(* IEC 61131-3 sources: dynamics/test, 21 files *)

(* ---- DeadbeatTest.st ---- *)
USING Simatic.Ax.Dynamics;
USING AxUnit;
USING System.Math;
NAMESPACE MyTest

    FUNCTION PT1 : LREAL
        VAR_INPUT
            t : LREAL;
            value : LREAL;
            output : LREAL;
            k : LREAL;
            t0 : LREAL;
        END_VAR
        PT1 := k * value + (output - k * value) * Exp(-1.0 * t / t0);
    END_FUNCTION

    {TestFixture}
    CLASS DeadbeatTest EXTENDS GlobalTest
        VAR
            controller : PT1_DeadbeatController;
        END_VAR

        {Test(k := 1, t0 := 1, output := 0, input := 0)}
        {Test(k := 1, t0 := 1, output := 0, input := 1)}
        {Test(k := 1, t0 := 1, output := 1, input := 0)}
        {Test(k := 1, t0 := 1, output := -78.5, input := 2.3)}
        {Test(k := 3.7, t0 := 5.8, output := -78.5, input := 2.3)}
        {Test(k := 107, t0 := 0.23, output := 10, input := 11)}
        METHOD PUBLIC Test
            VAR_INPUT
                k : LREAL;
                t0 : LREAL;
                output : LREAL;
                input : LREAL;
            END_VAR
            controller.SetK(k);
            controller.SetPeriods(oneSecondProvider.seconds, t0);
            Assert.Tolerated(input, PT1(oneSecondProvider.seconds, controller.Next(output, input), output, k, t0), TOLERANCE);
        END_METHOD
    END_CLASS
END_NAMESPACE

(* ---- Tolerated.st ---- *)
USING System.Math;
NAMESPACE AxUnit.Assert
    FUNCTION Tolerated
        VAR_INPUT
            expected : LREAL;
            actual : LREAL;
            tolerance : LREAL;
        END_VAR
        GreaterOrEqual(actual, expected - tolerance);
        LessOrEqual   (actual, expected + tolerance);
    END_FUNCTION
END_NAMESPACE

(* ---- AmplifierTest.st ---- *)
USING Simatic.Ax.Dynamics;

NAMESPACE MyTest
    {TestFixture}
    CLASS AmplifierTest EXTENDS GlobalTest

        VAR
            amplifier                   : Amplifier;
            value                       : ConstantSignal;
            expected                    : ConstantSignal;
        END_VAR

        // Amplifier
        {Test(k := 0, valueStepheight := 2.75)}
        {Test(k := 1, valueStepheight := 2.83)}
        {Test(k := 7.2, valueStepheight := 9.329)}
        {Test(k := 0.32, valueStepheight := 25.67)}
        METHOD PUBLIC Test
            VAR_INPUT
                k : LREAL;
                valueStepheight : LREAL;
            END_VAR
            amplifier.SetK(k);
            value.SetOutput(valueStepheight);
            expected.SetOutput(k * valueStepheight);
            THIS.AssertDynamic(expected, amplifier, value);
        END_METHOD

    END_CLASS
END_NAMESPACE

(* ---- BangBangTest.st ---- *)
USING Simatic.Ax.Dynamics;
USING AxUnit;

NAMESPACE MyTest
    {TestFixture}
    CLASS BangBangTest EXTENDS GlobalTest
        VAR
            controller : BangBangController;
        END_VAR

        // value0, value1, value2 and value3 are inside hysteresis
        {Test(input := 0, hysteresis := 1, output := FALSE, value0 := 0, value1 := 0, value2 := 0, value3 := 0)}
        {Test(input := 0, hysteresis := 1, output :=  TRUE, value0 := 0, value1 := 0, value2 := 0, value3 := 0)}
        {Test(input := 0, hysteresis := 1, output :=  TRUE, value0 := 0, value1 := -1, value2 := 1, value3 := 0.5)}
        {Test(input := 0, hysteresis := 10, output := FALSE, value0 := 2, value1 := -3, value2 := 5.7, value3 := -3.9)}
        {Test(input := 0, hysteresis := 83, output := TRUE, value0 := 20, value1 := -82.9, value2 := -83, value3 := 1.7)}
        METHOD PUBLIC TestWithinHysteresis
            VAR_INPUT
                input : LREAL;
                hysteresis: LREAL;
                output : BOOL;
                value0 : LREAL;
                value1 : LREAL;
                value2 : LREAL;
                value3 : LREAL;
            END_VAR
            controller.SetInput(input);
            controller.hysteresis := hysteresis;
            controller.SetOutput(output);
            Assert.Equal(controller.Next(value0), output);
            Assert.Equal(controller.Next(value1), output);
            Assert.Equal(controller.Next(value2), output);
            Assert.Equal(controller.Next(value3), output);
        END_METHOD

        // value is outside hysteresis
        {Test(input := 0,   hysteresis := 1,    heatingMode :=  TRUE, value := 2, expected := FALSE)}
        {Test(input := 0,   hysteresis := 1,    heatingMode := FALSE, value := 2, expected := TRUE)}
        {Test(input := 0,   hysteresis := 1,    heatingMode :=  TRUE, value := -2, expected := TRUE)}
        {Test(input := 0,   hysteresis := 1,    heatingMode := FALSE, value := -2, expected := FALSE)}
        {Test(input := 45,  hysteresis := 10,   heatingMode := FALSE, value := 34, expected := FALSE)}
        {Test(input := -3,  hysteresis := 0.1,  heatingMode := FALSE, value := -8, expected := FALSE)}
        {Test(input :=-107.59, hysteresis := 0, heatingMode := FALSE, value := -107.591, expected := FALSE)}
        {Test(input := 36.8, hysteresis := 2.5, heatingMode := FALSE, value := 31.8, expected := FALSE)}
        {Test(input := 45,  hysteresis := 10,   heatingMode :=  TRUE, value := 34, expected := TRUE)}
        {Test(input := -3,  hysteresis := 0.1,  heatingMode :=  TRUE, value := -8, expected := TRUE)}
        {Test(input :=-107.59, hysteresis := 0, heatingMode :=  TRUE, value := -107.591, expected := TRUE)}
        {Test(input := 36.8, hysteresis := 2.5, heatingMode :=  TRUE, value := 31.8, expected := TRUE)}
        {Test(input := 45,  hysteresis := 10,   heatingMode :=  TRUE, value := 56, expected := FALSE)}
        {Test(input := -3,  hysteresis := 0.1,  heatingMode :=  TRUE, value := -2, expected := FALSE)}
        {Test(input :=-107.59, hysteresis := 0, heatingMode :=  TRUE, value := -107.58, expected := FALSE)}
        {Test(input := 36.8, hysteresis := 2.5, heatingMode :=  TRUE, value := 41.8, expected := FALSE)}
        {Test(input := 45,  hysteresis := 10,   heatingMode := FALSE, value := 56, expected := TRUE)}
        {Test(input := -3,  hysteresis := 0.1,  heatingMode := FALSE, value := -2, expected := TRUE)}
        {Test(input :=-107.59, hysteresis := 0, heatingMode := FALSE, value := -107.58, expected := TRUE)}
        {Test(input := 36.8, hysteresis := 2.5, heatingMode := FALSE, value := 41.8, expected := TRUE)}
        METHOD PUBLIC TestOutsideHysteresis
            VAR_INPUT
                input : LREAL;
                hysteresis: LREAL;
                heatingMode : BOOL;
                value : LREAL;
                expected : BOOL;
            END_VAR
            controller.hysteresis := hysteresis;
            IF heatingMode THEN
                controller.EnableHeatingMode();
            ELSE
                controller.EnableCoolingMode();
            END_IF;
            Assert.Equal(controller.Next(value, input), expected);
        END_METHOD

    END_CLASS
END_NAMESPACE

(* ---- BoundedTest.st ---- *)
USING Simatic.Ax.Dynamics;
USING AxUnit;

NAMESPACE MyTest
    {TestFixture}
    CLASS BoundedTest EXTENDS GlobalTest
        VAR
            unboundedDynamic : IdentityDynamic;
            boundedDynamic   : BoundedDynamic;
        END_VAR

        {Test(value :=  0, observeMin := FALSE, minOutput := -1, observeMax := FALSE, maxOutput := 1, expected := 0)}
        {Test(value :=  0, observeMin :=  TRUE, minOutput := -1, observeMax := FALSE, maxOutput := 1, expected := 0)}
        {Test(value :=  0, observeMin := FALSE, minOutput := -1, observeMax :=  TRUE, maxOutput := 1, expected := 0)}
        {Test(value :=  0, observeMin :=  TRUE, minOutput := -1, observeMax :=  TRUE, maxOutput := 1, expected := 0)}
        {Test(value :=  2, observeMin := FALSE, minOutput := -1, observeMax := FALSE, maxOutput := 1, expected := 2)}
        {Test(value :=  2, observeMin :=  TRUE, minOutput := -1, observeMax := FALSE, maxOutput := 1, expected := 2)}
        {Test(value :=  2, observeMin := FALSE, minOutput := -1, observeMax :=  TRUE, maxOutput := 1, expected := 1)}
        {Test(value :=  2, observeMin :=  TRUE, minOutput := -1, observeMax :=  TRUE, maxOutput := 1, expected := 1)}
        {Test(value := -2, observeMin := FALSE, minOutput := -1, observeMax := FALSE, maxOutput := 1, expected := -2)}
        {Test(value := -2, observeMin :=  TRUE, minOutput := -1, observeMax := FALSE, maxOutput := 1, expected := -1)}
        {Test(value := -2, observeMin := FALSE, minOutput := -1, observeMax :=  TRUE, maxOutput := 1, expected := -2)}
        {Test(value := -2, observeMin :=  TRUE, minOutput := -1, observeMax :=  TRUE, maxOutput := 1, expected := -1)}
        {Test(value := -20.35, observeMin :=  TRUE, minOutput := -15.84, observeMax :=  TRUE, maxOutput := 1, expected := -15.84)}
        {Test(value := -20.35, observeMin :=  TRUE, minOutput := -65.84, observeMax :=  TRUE, maxOutput := -40, expected := -40)}
        METHOD PUBLIC Test
            VAR_INPUT
                value : LREAL;
                observeMin : BOOL;
                minOutput : LREAL;
                observeMax : BOOl;
                maxOutput  : LREAL;
                expected : LREAL;
            END_VAR
            boundedDynamic.unboundedDynamic := unboundedDynamic;
            boundedDynamic.observeMin := observeMin;
            boundedDynamic.minOutput := minOutput;
            boundedDynamic.observeMax := observeMax;
            boundedDynamic.maxOutput := maxOutput;
            Assert.Equal(expected, boundedDynamic.Next(value));
        END_METHOD

    END_CLASS
END_NAMESPACE

(* ---- ComposedOutputSignal.st ---- *)
USING Simatic.Ax.Dynamics;
NAMESPACE MyTest
    CLASS OutputComposedSignal IMPLEMENTS IOutputSignal
        VAR
            composedSignal : ComposedSignal;
            dynamic : IOutputDynamic;
        END_VAR

        METHOD PUBLIC SetInner
            VAR_INPUT
                newInner : ISignal;
            END_VAR
            composedSignal.inner := newInner;
        END_METHOD
        METHOD PUBLIC SetOuter
            VAR_INPUT
                newOuter : IOutputDynamic;
            END_VAR
            dynamic := newOuter;
            composedSignal.outer := newOuter;
        END_METHOD

        METHOD PUBLIC Next : LREAL
            Next := composedSignal.Next();
        END_METHOD

        METHOD PUBLIC GetOutput : LREAL
            GetOutput := dynamic.GetOutput();
        END_METHOD
    END_CLASS
END_NAMESPACE

(* ---- ComposedSignal.st ---- *)
USING Simatic.Ax.Dynamics;
NAMESPACE MyTest
    CLASS ComposedSignal IMPLEMENTS ISignal

        VAR PUBLIC
            inner : ISignal;
            outer : IDynamic;
        END_VAR

        METHOD PUBLIC Next : LREAL
            Next := outer.next(inner.Next());
        END_METHOD

    END_CLASS
END_NAMESPACE

(* ---- ConstantSignalTest.st ---- *)
USING AxUnit;
USING Simatic.Ax.Dynamics;

NAMESPACE MyTest
    {TestFixture}
    CLASS ConstantSignalTest EXTENDS GlobalTest
        VAR
            testerToTest : ConstantSignal;
        END_VAR
        {Test(output:=0)}
        {Test(output:=1)}
        {Test(output:=56.7)}
        {Test(output:=-23)}
        {Test(output:=-4.784)}
        METHOD PUBLIC Test
            VAR_INPUT
                output : LREAL;
            END_VAR
            testerToTest.output := output;
            Assert.Equal(output, testerToTest.Next());
            Assert.Equal(output, testerToTest.Next());
            Assert.Equal(output, testerToTest.Next());
        END_METHOD
    END_CLASS
END_NAMESPACE

(* ---- D_Test.st ---- *)
USING Simatic.Ax.Dynamics;

NAMESPACE MyTest
    {TestFixture}
    CLASS D_Test EXTENDS GlobalTest
        VAR
            value                       : RampSignal;
            expected                    : ConstantSignal;
            differentiator              : Differentiator;
        END_VAR

        {Test(valueSlope :=  1  , tD := 1)}
        // {Test(valueSlope :=  5.7, tD := 1.56)}
        // {Test(valueSlope := -3.8, tD := 2.37)}
        // {Test(valueSlope :=  104, tD := 43.1)}
        METHOD PUBLIC Test
            VAR_INPUT
                valueSlope : LREAL;
                tD : LREAL;
            END_VAR

            // Init value
            value.elapsedTimeProvider := oneSecondProvider;
            value.slope := valueSlope;

            // Init expected
            expected.output := valueSlope * tD;

            // Init differentiator
            differentiator.elapsedTimeProvider := oneSecondProvider;
            differentiator.SetTDSeconds(tD);

            // Assert
            THIS.AssertDynamic(expected, differentiator, value);
        END_METHOD

    END_CLASS
END_NAMESPACE

(* ---- DependentPaarallelSignal.st ---- *)
USING AxUnit;
USING Simatic.Ax.Dynamics;

NAMESPACE MyTest
    CLASS DependentParallelSignal IMPLEMENTS ISignal

        VAR PUBLIC
            independent : IOutputSignal;
            dependent : ISignal;
        END_VAR

        METHOD PUBLIC Next : LREAL
            Next := dependent.Next() + independent.GetOutput();
        END_METHOD

    END_CLASS
END_NAMESPACE

(* ---- DynamicControllerTest.st ---- *)
USING Simatic.Ax.Dynamics;
USING AxUnit;
NAMESPACE MyTest
    {TestFixture}
    CLASS DynamicCntrollerTest
        VAR
            amplifier : Amplifier;
            controller : DynamicController;
        END_VAR

        {Test(k := 1, input := 0, value := 0)}
        {Test(k := 1, input := 0, value := 1)}
        {Test(k := 1, input := 0, value := -1)}
        {Test(k := 1, input := 1, value := 0)}
        {Test(k := 1, input := -1, value := 0)}
        {Test(k := 5.7, input := 33.8, value := -3.4)}
        {Test(k := 3.7, input := -3.5, value := 83.4)}
        {Test(k := 310, input := 15.8, value := -0.1)}
        METHOD PUBLIC TestWithAmplifier
            VAR_INPUT
                k : LREAL;
                input : LREAL;
                value : LREAL;
            END_VAR
            amplifier.SetK(k);
            controller.openDynamic := amplifier;
            Assert.Equal(k * (input - value), controller.Next(value, input));
        END_METHOD
    END_CLASS
END_NAMESPACE

(* ---- GetSetTest.st ---- *)
USING TimeProviders;
USING Simatic.Ax.Dynamics;
USING AxUnit;
NAMESPACE MyTest
    {TestFixture}
    CLASS GetSetTest EXTENDS GlobalTest

        VAR
            amplifier : Amplifier;
            bangBangController : BangBangController;
            boundedDynamic : BoundedDynamic;
            boundedOutputDynamic : BoundedOutputDynamic;
            constantSignal : ConstantSignal;
            controller : DynamicController;
            differentiator : Differentiator;
            integrator : Integrator;
            pd_dynamic : PD_Dynamic;
            pi_dynamic : PI_Dynamic;
            pid_dynamic : PID_Dynamic;
            pt1_dynamic : PT1_Dynamic;
            pt1_deadbeatController : PT1_DeadbeatController;
            rampSignal : RampSignal;
        END_Var

        {Test(value := 0)}
        {Test(value := 1)}
        {Test(value := 2.7)}
        {Test(value := 83.9)}
        {Test(value := 475)}
        METHOD PUBLIC LRealTest
            VAR_INPUT
                value : LREAL;
            END_VAR

            amplifier.SetK(value);
            Assert.Equal(value, amplifier.GetK());

            bangBangController.SetInput(value);
            Assert.Equal(value, bangBangController.GetInput());

            boundedDynamic.SetMinOutput(value);
            Assert.Equal(value, boundedDynamic.GetMinOutput());
            boundedDynamic.SetMaxOutput(value);
            Assert.Equal(value, boundedDynamic.GetMaxOutput());

            boundedOutputDynamic.SetMinOutput(value);
            Assert.Equal(value, boundedOutputDynamic.GetMinOutput());
            boundedOutputDynamic.SetMaxOutput(value);
            Assert.Equal(value, boundedOutputDynamic.GetMaxOutput());

            constantSignal.SetOutput(value);
            Assert.Equal(value, constantSignal.GetOutput());

            controller.SetInput(value);
            Assert.Equal(value, controller.GetInput());

            differentiator.SetTDSeconds(value);
            Assert.Equal(value, differentiator.GetTDSeconds());

            integrator.SetTISeconds(value);
            Assert.Equal(value, integrator.GetTISeconds());
            integrator.SetOutput(value);
            Assert.Equal(value, integrator.GetOutput());

            pd_dynamic.SetK(value);
            Assert.Equal(value, pd_dynamic.GetK());
            pd_dynamic.SetTDSeconds(value);
            Assert.Equal(value, pd_dynamic.GetTDSeconds());

            pi_dynamic.SetK(value);
            Assert.Equal(value, pi_dynamic.GetK());
            pi_dynamic.SetTISeconds(value);
            Assert.Equal(value, pi_dynamic.GetTISeconds());

            pid_dynamic.SetK(value);
            Assert.Equal(value, pid_dynamic.GetK());
            pid_dynamic.SetTISeconds(value);
            Assert.Equal(value, pid_dynamic.GetTISeconds());
            pid_dynamic.SetTDSeconds(value);
            Assert.Equal(value, pid_dynamic.GetTDSeconds());
            pid_dynamic.SetIntegratorMinOutput(value);
            Assert.Equal(value, pid_dynamic.GetIntegratorMinOutput());
            pid_dynamic.SetIntegratorMaxOutput(value);
            Assert.Equal(value, pid_dynamic.GetIntegratorMaxOutput());

            pt1_dynamic.SetK(value);
            Assert.Equal(value, pt1_dynamic.GetK());
            pt1_dynamic.SetT0Seconds(value);
            Assert.Equal(value, pt1_dynamic.GetT0Seconds());

            pt1_deadbeatController.SetK(value);
            Assert.Equal(value, pt1_deadbeatController.GetK());

            rampSignal.SetTISeconds(value);
            Assert.Equal(value, rampSignal.GetTISeconds());
            rampSignal.SetOutput(value);
            Assert.Equal(value, rampSignal.GetOutput());
        END_METHOD

        {Test(value0 := 1, value1 := 1)}
        {Test(value0 := 2.8, value1 := 29.5)}
        {Test(value0 := 6.54, value1 := 0.3)}
        METHOD PUBLIC LRealsTest
            VAR_INPUT
                value0 : LREAL;
                value1 : LREAL;
            END_VAR

            differentiator.SetTDSeconds(value0, value1);
            Assert.Equal(value0 * value1, differentiator.GetTDSeconds());

            integrator.SetTISeconds(value0, value1);
            Assert.Equal(value0 / value1, integrator.GetTISeconds());
        END_METHOD

        {Test(value := FALSE)}
        {Test(value := TRUE)}
        METHOD PUBLIC BooleanTest
            VAR_INPUT
                value : BOOL;
            END_VAR

            IF value THEN
                bangBangController.EnableHeatingMode();
            ELSE
                bangBangController.EnableCoolingMode();
            END_IF;
            Assert.Equal(    value, bangBangController.IsHeatingModeEnabled());
            Assert.Equal(NOT value, bangBangController.IsCoolingModeEnabled());

            bangBangController.SetOutput(value);
            Assert.Equal(value, bangBangController.GetOutput());
        END_METHOD
    END_CLASS
END_NAMESPACE

(* ---- GlobalTest.st ---- *)
USING TimeProviders;
USING Simatic.Ax.Dynamics;
USING AxUnit;

NAMESPACE MyTest
    CLASS GlobalTest

        VAR CONSTANT
            TOLERANCE                   : LREAL := 1.0e-5;
            DURATION                    : UINT := UINT#12;
        END_VAR
        VAR PROTECTED
            oneSecondProvider           : ConstantTimeProvider := (seconds := 1.0);
        END_VAR
        VAR PRIVATE
            _actual                      : ComposedSignal;
        END_VAR

        METHOD AssertSignal
            VAR_INPUT
                expected : ISignal;
                actual : ISignal;
            END_VAR
            VAR_TEMP
                cycle : UINT;
            END_VAR
            FOR cycle := UINT#1 TO DURATION DO
                Assert.Tolerated(expected.Next(), actual.Next(), TOLERANCE);
            END_FOR;
        END_METHOD

        METHOD AssertDynamic
            VAR_INPUT
                expected : ISignal;
                dynamic : IDynamic;
                value : ISignal;
            END_VAR
            _actual.inner := value;
            _actual.outer := dynamic;
            THIS.AssertSignal(expected, _actual);
        END_METHOD

    END_CLASS
END_NAMESPACE

(* ---- I_Test.st ---- *)
USING Simatic.Ax.Dynamics;

NAMESPACE MyTest
    {TestFixture}
    CLASS I_Test EXTENDS GlobalTest
        VAR
            value                       : ConstantSignal;
            expected                    : RampSignal;
            integrator                  : Integrator;
        END_VAR

        {Test(valueStepheight :=  1.0, t := 1)}
        {Test(valueStepheight :=  5.7, t := 1.56)}
        {Test(valueStepheight := -3.8, t := 2.37)}
        {Test(valueStepheight :=  104, t := 43.1)}
        METHOD PUBLIC Test
            VAR_INPUT
                valueStepheight : LREAL;
                t : LREAL;
            END_VAR

            // Init value
            value.output := valueStepheight;

            // Init expected
            expected.elapsedTimeProvider := oneSecondProvider;
            expected.SetTISeconds(t / valueStepheight);

            // Init integrator
            integrator.elapsedTimeProvider := oneSecondProvider;
            integrator.SetTISeconds(t);

            // Assert
            THIS.AssertDynamic(expected, integrator, value);
        END_METHOD

    END_CLASS
END_NAMESPACE

(* ---- ParallelSignal.st ---- *)
USING AxUnit;
USING Simatic.Ax.Dynamics;

NAMESPACE MyTest
    CLASS ParallelSignal IMPLEMENTS ISignal

        VAR PUBLIC
            signal0 : ISignal;
            signal1 : ISignal;
        END_VAR

        METHOD PUBLIC Next : LREAL
            Next := signal0.Next() + signal1.Next();
        END_METHOD

    END_CLASS
END_NAMESPACE

(* ---- PD_Test.st ---- *)
USING Simatic.Ax.Dynamics;
USING AxUnit.Assert;

NAMESPACE MyTest
    {TestFixture}
    CLASS PD_Test EXTENDS GlobalTest
        VAR
            value                       : RampSignal;
            step                        : ConstantSignal;
            ramp                        : RampSignal;
            expected                    : ParallelSignal;
            dynamic                     : PD_Dynamic;
        END_VAR

        {Test(slope :=  1.0, k :=   1   , t := 1)}
        {Test(slope :=  2.0, k :=   1   , t := 1)}
        {Test(slope :=  1.0, k :=   2   , t := 1)}
        {Test(slope :=  1.0, k :=   1   , t := 2)}
        {Test(slope :=  5.7, k :=   0.23, t := 1.56)}
        {Test(slope := -3.8, k :=   9.74, t := 2.37)}
        {Test(slope :=  104, k := -34.81, t := 43.1)}
        METHOD PUBLIC Test
            VAR_INPUT
                slope : LREAL;
                k : LREAL;
                t : LREAL;
            END_VAR

            // Init value
            value.elapsedTimeProvider := oneSecondProvider;
            value.slope := slope;

            // Init step
            step.output := k * slope * t;

            // Init ramp
            ramp.elapsedTimeProvider := oneSecondProvider;
            ramp.slope := k * slope;

            // Init expected
            expected.signal0 := step;
            expected.signal1 := ramp;

            // Init dynamic
            dynamic.elapsedTimeProvider := oneSecondProvider;
            dynamic.SetK(k);
            dynamic.SetTDSeconds(t);

            // Assert
            THIS.AssertDynamic(expected, dynamic, value);
        END_METHOD

    END_CLASS
END_NAMESPACE

(* ---- PI_Test.st ---- *)
USING Simatic.Ax.Dynamics;
USING AxUnit.Assert;

NAMESPACE MyTest
    {TestFixture}
    CLASS PI_Test EXTENDS GlobalTest
        VAR
            value                       : ConstantSignal;
            step                        : ConstantSignal;
            ramp                        : RampSignal;
            expected                    : ParallelSignal;
            dynamic                     : PI_Dynamic;
        END_VAR

        {Test(valueStepheight :=  1.0, k :=   1   , t := 1)}
        {Test(valueStepheight :=  5.7, k :=   0.23, t := 1.56)}
        {Test(valueStepheight := -3.8, k :=   9.74, t := 2.37)}
        {Test(valueStepheight :=  104, k := -34.81, t := 43.1)}
        METHOD PUBLIC Test
            VAR_INPUT
                valueStepheight : LREAL;
                k : LREAL;
                t : LREAL;
            END_VAR

            // Init value
            value.output := valueStepheight;

            // Init step
            step.output := k * valueStepheight;

            // Init ramp
            ramp.elapsedTimeProvider := oneSecondProvider;
            ramp.slope := k * valueStepheight / t;

            // Init expected
            expected.signal0 := step;
            expected.signal1 := ramp;

            // Init dynamic
            dynamic.elapsedTimeProvider := oneSecondProvider;
            dynamic.SetK(k);
            dynamic.SetTISeconds(t);

            // Assert
            THIS.AssertDynamic(expected, dynamic, value);
        END_METHOD

    END_CLASS
END_NAMESPACE

(* ---- PID_RampResponse.st ---- *)
USING Simatic.Ax.Dynamics;

NAMESPACE MyTest
    CLASS PID_RampResponse EXTENDS ExplicitSignal

        VAR PUBLIC
            k : LREAL;
            tISeconds : LREAL;
            tDSeconds : LREAL;
        END_VAR

        METHOD PROTECTED OVERRIDE _GetOutput : LREAL
            VAR_INPUT
                cycle : UINT;
            END_VAR
            _GetOutput := k * (
                cycle +
                cycle * (cycle + 1.0) / 2.0 / tISeconds +
                tDSeconds
            );
        END_METHOD

    END_CLASS
END_NAMESPACE

(* ---- PID_Test.st ---- *)
USING Simatic.Ax.Dynamics;

NAMESPACE MyTest
    {TestFixture}
    CLASS PID_Test EXTENDS GlobalTest

        VAR
            expected : PID_RampResponse;
            dynamic : PID_Dynamic;
            value : RampSignal;
        END_VAR

        {Test(k := 1, td := 1, ti := 1)}
        // {Test(k := 2, td := 1, ti := 1)}
        // {Test(k := 1, td := 2, ti := 1)}
        // {Test(k := 1, td := 1, ti := 2)}
        // {Test(k := 3.7, td := 5.3, ti := 0.28)}
        // {Test(k := -1.7, td := 0.39, ti := 5.6)}
        METHOD PUBLIC Test_d_pi
            VAR_INPUT
                k: LREAL;
                tD: LREAL;
                tI: LREAL;
            END_VAR

            // Init expected
            expected.k := k;
            expected.tDSeconds := tD;
            expected.tISeconds := tI;

            // Init dynamic
            dynamic.elapsedTimeProvider := oneSecondProvider;
            dynamic.setK(k);
            dynamic.SetTDSeconds(tD);
            dynamic.SetTISeconds(tI);

            // Init value
            value.elapsedTimeProvider := oneSecondProvider;
            value.slope := 1.0;

            // Assert
            THIS.AssertDynamic(expected, dynamic, value);
        END_METHOD

    END_CLASS
END_NAMESPACE

(* ---- PT1_Test.st ---- *)
USING AxUnit;
USING Simatic.Ax.Dynamics;
USING AxUnit;

NAMESPACE MyTest
    {TestFixture}
    CLASS PT1_Test EXTENDS GlobalTest

        VAR
            dynamic : PT1_Dynamic;
        END_VAR

        {Test(valueStepheight :=  1.0, k :=   1   , t0 := 1)}
        {Test(valueStepheight :=  2.0, k :=   1   , t0 := 1)}
        {Test(valueStepheight :=  1.0, k :=   2   , t0 := 1)}
        {Test(valueStepheight :=  1.0, k :=   1   , t0 := 2)}
        {Test(valueStepheight :=  5.7, k :=   0.23, t0 := 100)}
        {Test(valueStepheight := -3.8, k :=   9.74, t0 := 12)}
        {Test(valueStepheight :=  104, k := -34.81, t0 := 60)}
        METHOD PUBLIC Test
            VAR_INPUT
                k : LREAL;
                t0 : LREAL;
                valueStepheight : LREAL;
            END_VAR

            // Init dynamic
            dynamic.elapsedTimeProvider := oneSecondProvider;
            dynamic.SetK(k);
            dynamic.SetT0Seconds(t0);

            Assert.Tolerated(k * valueStepheight / t0, dynamic.Next(valueStepheight), TOLERANCE);
        END_METHOD

    END_CLASS
END_NAMESPACE

(* ---- RampTest.st ---- *)
USING AxUnit;
USING Simatic.Ax.Dynamics;

NAMESPACE MyTest
    {TestFixture}
    CLASS RampTest EXTENDS GlobalTest

        VAR
            actual : RampSignal;
        END_VAR

        {Test(slope := 1)}
        {Test(slope := -2.7)}
        {Test(slope := 1.3)}
        METHOD PUBLIC SlopeTest
            VAR_INPUT
                slope : LREAL;
            END_VAR
            actual.slope := slope;
            actual.elapsedTimeProvider := oneSecondProvider;
            Assert.Equal(slope, actual.Next());
            Assert.Tolerated(2*slope, actual.Next(), TOLERANCE);
            Assert.Tolerated(3*slope, actual.Next(), TOLERANCE);
            Assert.Tolerated(4*slope, actual.Next(), TOLERANCE);
        END_METHOD

        {Test(tI := 1)}
        {Test(tI := -2.7)}
        {Test(tI := 1.3)}
        METHOD PUBLIC TITest
            VAR_INPUT
                tI : LREAL;
            END_VAR
            actual.SetTISeconds(tI);
            actual.elapsedTimeProvider := oneSecondProvider;
            Assert.Tolerated(1/tI, actual.Next());
            Assert.Tolerated(2/tI, actual.Next(), TOLERANCE);
            Assert.Tolerated(3/tI, actual.Next(), TOLERANCE);
            Assert.Tolerated(4/tI, actual.Next(), TOLERANCE);
        END_METHOD

    END_CLASS
END_NAMESPACE
